PROGRAM MAIN
VAR
	
	BasicTestingEnabled					: BOOL;
                            			
	FB_BlindControl						: ARRAY [0..2] OF BlindControl;
                            			
	i									: INT;
                            			
	bTest								: BOOL;
	bLog								: BOOL;
                    					
	arrData								: ARRAY[0..BUFFER_SIZE] OF ST_PHASE_DATA;
	arrSnapshotData						: ARRAY[0..BUFFER_SIZE] OF ST_PHASE_DATA;
                    					
	iState								: INT;
	bExecute							: BOOL;
	bBusy								: BOOL;
                            	
	bError 								: BOOL;
	tonSampleRate						: TON;

	aDataPacket1						: ARRAY [0..6] OF BYTE := [16#9A, 16#04, 16#00, 16#00, 16#0A, 16#00, 16#00]; 		(* Main office *)
	aDataPacket2						: ARRAY [0..6] OF BYTE :=  [16#9A, 16#02, 16#00, 16#00, 16#0A, 16#00, 16#00];		(* Board Room*)
	aDataPacket3						: ARRAY [0..6] OF BYTE := [16#9A, 16#03, 16#00, 16#00, 16#0A, 16#00, 16#00]; 		(* Reception *)
	
	
	bStretch							: BOOL;
	bStretchDone						: BOOL;
	HowOftenTimer						: Ton := (PT:= T#21d);//31d);
		
	fbBlindsStretch						: BlindStretch;

	hmiStrech							: BOOL;
	
	fbWindSimulator						: FB_WindTurbineSim;
	
	windSpeed							: LREAL;
	
	bGetOpenWeatherMap             		: BOOL;

    fbHttpClientOpenWeatherMap     		: FB_IotHttpClient :=(sHostName:='api.weatherapi.com', bKeepAlive:=TRUE, tConnectionTimeout:=T#10S);

    fbWeatherAPI        				: FB_WeatherAPI_HTTP;
	
	fbSendWatsappCallMeBot				: FB_SendWhatsappCallMeBot;
	
	fbHttpClientWhatsAppResponse   		: FB_IotHttpClient :=(sHostName:='webhook.site', bKeepAlive:=TRUE, tConnectionTimeout:=T#10S);
	
	fbWhatsAppRespose					: FB_WatsAppResponse;
	
	textWhatsApp						: T_MaxString;
	
	weatherTon							: ton := (pt:=T#10m);					
	local: BOOL;
	hmiFinished: BOOL;
	testWhatsApp: BOOL;
END_VAR

BackgroundComms();
ADSReadCX9020();
EnOcean();
//SQLDB();
PrgMqttCom_PM_Subscriber();
//PrgMqttCom_Blinds_Publisher();
//CoffeePredictionML();
//MLtest();
Dali();
//DMX();
LightControl();
//ReadCP67();
FileHandle();
TableTennisScoreCounter();
VariableHandleForHmi();
SleepModeCheck();
PowerSupply();

FB_BlindControl[0](
	BulkCommand:= BackgroundComms.BlindCommandTable[0].SelectBlindsBulkCommand ,
	xCommandUp:= BackgroundComms.BlindCommandTable[0].xCommandUp,
	xCommandDown:= BackgroundComms.BlindCommandTable[0].xCommandDown ,
	xCommandStop:= BackgroundComms.BlindCommandTable[0].xCommandStop ,
	HubTXBuffer:= BackgroundComms.HubTXBuffer[0] ,
	HubRXBuffer:= BackgroundComms.HubRXBuffer[0] ,
	aDataPacket := aDataPacket1,
	xCommandUpJog := BackgroundComms.BlindCommandTable[0].xCommandUpJog ,
	xCommandDownJog := BackgroundComms.BlindCommandTable[0].xCommandDownJog ,
	JogTime :=  BackgroundComms.BlindCommandTable[0].JogTime,
	JogTimeInt :=  BackgroundComms.BlindCommandTable[0].JogTimeInt,
	xBusy => );

FB_BlindControl[1](
	BulkCommand:= BackgroundComms.BlindCommandTable[1].SelectBlindsBulkCommand ,
	xCommandUp:= BackgroundComms.BlindCommandTable[1].xCommandUp,
	xCommandDown:= BackgroundComms.BlindCommandTable[1].xCommandDown ,
	xCommandStop:= BackgroundComms.BlindCommandTable[1].xCommandStop ,
	HubTXBuffer:= BackgroundComms.HubTXBuffer[1] ,
	HubRXBuffer:= BackgroundComms.HubRXBuffer[1] ,
	aDataPacket :=  aDataPacket2,
	xCommandUpJog := BackgroundComms.BlindCommandTable[1].xCommandUpJog ,
	xCommandDownJog := BackgroundComms.BlindCommandTable[1].xCommandDownJog ,
	JogTime :=  BackgroundComms.BlindCommandTable[1].JogTime,
	JogTimeInt :=  BackgroundComms.BlindCommandTable[1].JogTimeInt,
	xBusy => );

FB_BlindControl[2](
	BulkCommand:= BackgroundComms.BlindCommandTable[2].SelectBlindsBulkCommand ,
	xCommandUp:= BackgroundComms.BlindCommandTable[2].xCommandUp,
	xCommandDown:= BackgroundComms.BlindCommandTable[2].xCommandDown ,
	xCommandStop:= BackgroundComms.BlindCommandTable[2].xCommandStop ,
	HubTXBuffer:= BackgroundComms.HubTXBuffer[2] ,
	HubRXBuffer:= BackgroundComms.HubRXBuffer[2] ,
	aDataPacket :=  aDataPacket3,
	xCommandUpJog := BackgroundComms.BlindCommandTable[2].xCommandUpJog ,
	xCommandDownJog := BackgroundComms.BlindCommandTable[2].xCommandDownJog ,
	JogTime :=  BackgroundComms.BlindCommandTable[2].JogTime,
	JogTimeInt :=  BackgroundComms.BlindCommandTable[2].JogTimeInt,
	xBusy => );
	

HowOftenTimer.IN:= TRUE;

IF HowOftenTimer.Q THEN
	bStretch := TRUE;
	hmiFinished := FALSE;
END_IF

IF bStretchDone THEN
	HowOftenTimer.IN := FALSE;
	bStretchDone := FALSE;
	bStretch := FALSE;
	hmiStrech := FALSE;
	hmiFinished := TRUE;
END_IF
	
fbBlindsStretch(Start:= bStretch AND hmiStrech, StretchDone:= bStretchDone,Err=> );

HowOftenTimer();

IF NOT fbHttpClientOpenWeatherMap.bConfigured THEN
    fbHttpClientOpenWeatherMap.nHostPort:= 443;
    fbHttpClientOpenWeatherMap.stTLS.bNoServerCertCheck:= TRUE;
	weatherTon.IN := TRUE;
END_IF

IF fbHttpClientOpenWeatherMap.bConfigured THEN
    fbWeatherAPI(bSend:=weatherTon.Q, fbClient:=fbHttpClientOpenWeatherMap);
END_IF

IF weatherTon.Q THEN
	weatherTon.IN := FALSE;
ELSE
	weatherTon.IN := TRUE;
END_IF

fbHttpClientOpenWeatherMap.Execute();
WindSpeed := fbWeatherAPI.wind_speed;
fbWindSimulator(windSpeed:= WindSpeed, rpm=> RPM, powerOutput=> Power);
weatherTon();

fbSendWatsappCallMeBot(SendText := , YourNumber := '447724278323', Text2Send := textWhatsApp, ApiKey := '6082625');  //SendText := , YourNumber := '+447724278323', Text2Send := textWhatsApp, ApiKey := 'US6Y79pt7LAU'

IF testWhatsApp THEN	//RPM > 200 AND weatherTon.Q 
	textWhatsApp := 'Wind turbine at risk, consider switching the turbine off.';
	fbSendWatsappCallMeBot.SendText := TRUE;
ELSE
	fbSendWatsappCallMeBot.SendText := FALSE;
END_IF

IF NOT fbHttpClientWhatsAppResponse.bConfigured THEN
    fbHttpClientOpenWeatherMap.nHostPort:= 443;
    fbHttpClientOpenWeatherMap.stTLS.bNoServerCertCheck:= TRUE;
	//weatherTon.IN := TRUE;
END_IF

IF fbHttpClientWhatsAppResponse.bConfigured THEN
    fbWhatsAppRespose(bSend:=testWhatsApp, fbClient:=fbHttpClientWhatsAppResponse);
END_IF

fbHttpClientWhatsAppResponse.Execute();

ACTION SleepModeCheck:
IF Global_Variables.xSleepMode THEN
	
	// Set Socket State
	xXplanarScreenPowerOff := TRUE;
	
		

	xSleepMode := FALSE;						// Reset Sleep Call	
	
END_IF
END_ACTION

END_PROGRAM

(* stored: Version 1.1.0.1, ProductVersion 3.1.4024.12
   POU MAIN: Id {a3e1c45b-7b61-493c-b315-876295153612}, SpecialFunc None
   Action SleepModeCheck: Id {3f87cb06-794c-44e6-adeb-1113c47adff4} *)
